SUBAPPLICATION Uebung_029 (* LED_DO Blinkende LED *)
  (* Standard: 61499-2 *)
  (* Version 1.0, 2023-10-23, franz *)
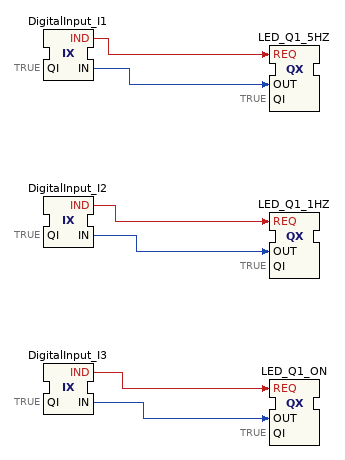
  FBS
    LED_Q1_5HZ : QX(QI := TRUE);
    DigitalInput_I1 : IX(QI := TRUE);
    LED_Q1_1HZ : QX(QI := TRUE);
    DigitalInput_I2 : IX(QI := TRUE);
    LED_Q1_ON : QX(QI := TRUE);
    DigitalInput_I3 : IX(QI := TRUE);
  END_FBS
  EVENT_CONNECTIONS
    DigitalInput_I1.IND TO LED_Q1_5HZ.REQ;
    DigitalInput_I2.IND TO LED_Q1_1HZ.REQ;
    DigitalInput_I3.IND TO LED_Q1_ON.REQ;
  END_CONNECTIONS
  DATA_CONNECTIONS
    DigitalInput_I1.IN TO LED_Q1_5HZ.OUT;
    DigitalInput_I2.IN TO LED_Q1_1HZ.OUT;
    DigitalInput_I3.IN TO LED_Q1_ON.OUT;
  END_CONNECTIONS
END_SUBAPPLICATION
